// TIA Portal V17 export
// export: Created 2024-01-30T08:49:16.4839572Z, ExportSetting WithDefaults, DisplayName Totally Integrated Automation Portal, DisplayVersion V17 Update 6, DisplayName TIA Portal Openness, DisplayVersion V17 Update 6, DisplayName TIA Portal Version Control Interface, DisplayVersion V17, DisplayName STEP 7 Professional, DisplayVersion V17 Update 6, DisplayName STEP 7 Safety, DisplayVersion V17 Update 6, DisplayName WinCC Advanced, DisplayVersion V17 Update 6
DATA_BLOCK "R_TRIG_DB"   // DB19
// stored: AutoNumber true, DBAccessibleFromOPCUA true, DBAccessibleFromWebserver true, InstanceOfName R_TRIG, OfSystemLibElement R_TRIG, OfSystemLibVersion 1.0
"R_TRIG"
   // VAR_INPUT
   //    CLK : Bool;
   // END_VAR
   // VAR_OUTPUT
   //    Q : Bool;
   // END_VAR
   // VAR
   //    Stat_Bit : Bool;
   // END_VAR
BEGIN
END_DATA_BLOCK
